(* PLC project Generated.project, CODESYS CODESYS V3.5 SP19 Patch 1 *)
(* stored: creationDateTime 2026-09-06T13:00:42.469933, modificationDateTime 2026-09-06T13:00:42.469933 *)

(* ═══════════════════════════════════════════════════════════════ ST_SyncCfg — Configuration de la synchronisation M1/M2 ═══════════════════════════════════════════════════════════════ *)
TYPE ST_SyncCfg : STRUCT
  CfgSyncTolerance_M : REAL := 3;  (* 📐 Tolérance max d'écart (m) — Dégradation Palier 1 dès 3.0m *)
  CfgSyncCriticalTolerance_M : REAL := 6;  (* 🔴 Seuil 2 critique (m) — blocage synchro ; doit être > CfgSyncTolerance_M *)
  Initialized : BOOL := FALSE;  (* 🚦 Flag restauration boot (config restaurée depuis GVL_PERSISTENT) *)
END_STRUCT;
END_TYPE

(* ======================================================================= 💾 FB_CfgPersistBridge_SyncCfg — Pont persistance pour ST_SyncCfg ─────────────────────────────────────────────────────────────── 🎯 Rôle : Restauration et synchronisation bidirectionnelle IHM / Persist 💾 Persistance : Transfert GVL_PERSISTENT <-> GVL_IHM sur Initialized 📄 Doc métier : DOC/AF/AF_Partie-03_Contrats_Composants_v2.3.md §3 ======================================================================= *)
FUNCTION_BLOCK FB_CfgPersistBridge_SyncCfg
  VAR_OUTPUT
    JustRestored : BOOL;  (* === ETATS RESTAURATION === <-- [STAT] Vrai sur le cycle de restauration initiale *)
  END_VAR
  VAR_IN_OUT
    Hmi : ST_SyncCfg;  (* === BUS CONFIGURATION ET PERSISTANCE === <-> [BUS] Structure de configuration IHM *)
    Persist : ST_SyncCfg;  (* <-> [BUS] Structure de configuration persistante *)
  END_VAR

            

JustRestored := FALSE;
IF NOT Hmi.Initialized THEN
    Hmi := Persist;
    Hmi.Initialized := TRUE;
    JustRestored := TRUE;
ELSE
    Persist := Hmi;
END_IF;

          
END_FUNCTION_BLOCK
